FUNCTION_BLOCK CLIENT_1_6 (* 1-Input,6-Output Client Interface *)
  (* Standard: 61499-1; Classification: Communications *)
  (* Version 0.0, 2005-06-10, JHC, Holobloc Inc *)
  (* Compiler header: package fb.rt.net; *)
  (* Compiler Java Sun JDK 1.5.0 *)
  (* Compiler Java IBM VisualAge 3.0 *)
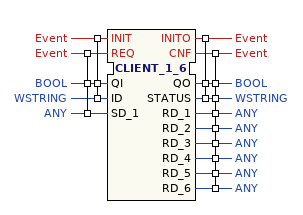
  EVENT_INPUT
    INIT WITH QI, ID; (* Service Initialization *)
    REQ WITH QI, SD_1; (* Service Request *)
  END_EVENT
  EVENT_OUTPUT
    INITO WITH QO, STATUS; (* Initialization Confirm *)
    CNF WITH QO, STATUS, RD_1, RD_2, RD_3, RD_4, RD_5, RD_6; (* Service Confirmation *)
  END_EVENT
  VAR_INPUT
    QI : BOOL; (* Event Input Qualifier *)
    ID : WSTRING; (* Connection Identifier *)
    SD_1 : ANY; (* Data to Send *)
  END_VAR
  VAR_OUTPUT
    QO : BOOL; (* Event Output Qualifier *)
    STATUS : WSTRING; (* Service Status *)
    RD_1 : ANY; (* Received Data *)
    RD_2 : ANY; (* Received Data *)
    RD_3 : ANY; (* Received Data *)
    RD_4 : ANY; (* Received Data *)
    RD_5 : ANY; (* Received Data *)
    RD_6 : ANY; (* Received Data *)
  END_VAR
END_FUNCTION_BLOCK
